(* IEC 61131-3 sources: SigmatekTestframework/src/Class/CExternalTest, 1 file *)

(* ---- CExternalTest.st ---- *)
(*!
<Class
	Name               = "CExternalTest"
	Revision           = "1.1"
	RealtimeTask       = "false"
	CyclicTask         = "false"
	BackgroundTask     = "false"
	Sigmatek           = "false"
	OSInterface        = "false"
	HighPriority       = "false"
	Automatic          = "false"
	UpdateMode         = "Prescan"
	SharedCommandTable = "true"
	Objectsize         = "(284,120)"
	Singleton          = "true">
	<Channels>
		<Server Name="State" Visualized="false" Initialize="false" WriteProtected="true" Retentive="false"/>
		<Client Name="Finished" Required="true" Internal="false"/>
		<Client Name="Start" Required="true" Internal="false"/>
	</Channels>
	<Network Name="CExternalTest">
		<!-- List of Components in this network -->
		<Components>
		</Components>
		<Comments>
		</Comments>
		<!-- List of Connections in this network -->
		<Connections>
		</Connections>
		<!-- Headerfiles -->
		<Options>
		</Options>
	</Network>
</Class>
*)
CExternalTest : CLASS
  //Servers:
	State 	: SvrChCmd_DINT;
  //Clients:
	Start 	: CltCh_DINT;
	Finished 	: CltCh_DINT;
  //Variables:
		m_pLib 	: ^CTestLib;
  //Functions:

	FUNCTION VIRTUAL GLOBAL Init;
				//! <Function Comment="optional method&#13;&#10;called before execute" Name="prepare"/>
	FUNCTION VIRTUAL GLOBAL prepare
		VAR_OUTPUT
			bRetcode 	: BOOL;
		END_VAR;
				//! <Function Comment="execute test" Name="execute"/>
	FUNCTION VIRTUAL GLOBAL execute
		VAR_OUTPUT
			bRetcode 	: BOOL;
		END_VAR;
				//! <Function Comment="optional method&#13;&#10;called after execute" Name="cleanUp"/>
	FUNCTION VIRTUAL GLOBAL cleanUp
		VAR_OUTPUT
			bRetcode 	: BOOL;
		END_VAR;
  //Tables:
	FUNCTION @STD
		VAR_OUTPUT
			ret_code	: CONFSTATES;
		END_VAR;
	FUNCTION GLOBAL TAB @CT_;
END_CLASS;

#pragma usingLtd CTestLib

//Exclude-SccX
(*
 **********************************************************************
 * \file CExternalTest.st
 *
 * Dummy Class to use other Testframeworks
 *
 * Copyright (c) 2023,Hoox.Software, Helmbrechts
 * All Rights Reserved.
 *
 * Created on: 22.03.2023
 *     Author: dressel
 *
 **********************************************************************
 *)

//*********************************************************************
//
//
//*********************************************************************
FUNCTION VIRTUAL GLOBAL CExternalTest::Init

   if _FirstScan then

      State := 0;

      m_pLib := _LookUpObj(pName:= "TestLib")$^CTestLib;

      if m_pLib <> nil then
         if m_pLib^.registerExternalTest(this) = false then
            State := -1;
         else
            State := 1;
         end_if;
      end_if;

   end_if;

END_FUNCTION

//*********************************************************************
//
//
//*********************************************************************
FUNCTION VIRTUAL GLOBAL CExternalTest::prepare
	VAR_OUTPUT
		bRetcode 	: BOOL;
	END_VAR

   Start := 1;
   Start.Write(Start);

   bRetcode := true;

END_FUNCTION

//*********************************************************************
//
//
//*********************************************************************
FUNCTION VIRTUAL GLOBAL CExternalTest::execute
	VAR_OUTPUT
		bRetcode 	: BOOL;
	END_VAR

   Finished := Finished.Read();
   bRetcode := (Finished <> 0);

END_FUNCTION

//*********************************************************************
//
//
//*********************************************************************
FUNCTION VIRTUAL GLOBAL CExternalTest::cleanUp
	VAR_OUTPUT
		bRetcode 	: BOOL;
	END_VAR

   Start := 0;
   Start.Write(Start);

   bRetcode := true;

END_FUNCTION
